//
// Currently unsupported types:
//
// ADSDATATYPEID.ADST_BIGTYPE;
// ADSDATATYPEID.ADST_REAL80;
// ADSDATATYPEID.ADST_VOID;
// ADSDATATYPEID.ADST_STRING
// ADSDATATYPEID.ADST_WSTRING

FUNCTION F_ParseToVariant : bool
VAR_INPUT
	adsTypeID  : ADSDATATYPEID;
	sValue		 : STRING;
END_VAR
VAR_IN_OUT
		var_data : ST_VARIANT;
END_VAR


	F_ParseToVariant:= TRUE;	
	
	CASE adsTypeID OF 
		
		ADSDATATYPEID.ADST_INT8:
			var_data.nI8 := STRING_TO_SINT(sValue);

		ADSDATATYPEID.ADST_UINT8:
			var_data.nUI8 := STRING_TO_USINT(sValue);
					
		ADSDATATYPEID.ADST_INT16:
			var_data.nI16 := STRING_TO_INT(sValue);
		
		ADSDATATYPEID.ADST_UINT16:
			var_data.nUI16 := STRING_TO_UINT(sValue);
						
		ADSDATATYPEID.ADST_INT32:
			var_data.nI32 := STRING_TO_DINT(sValue);

		ADSDATATYPEID.ADST_UINT32:
			var_data.nUI32 := STRING_TO_UDINT(sValue);
			
		ADSDATATYPEID.ADST_INT64:
			var_data.nI64 := STRING_TO_LINT(sValue);

		ADSDATATYPEID.ADST_UINT64:
			var_data.nUI64 := STRING_TO_ULINT(sValue);			

		ADSDATATYPEID.ADST_REAL32:
			var_data.fR32 := STRING_TO_REAL(sValue);
						
		ADSDATATYPEID.ADST_REAL64:
			var_data.fR64 := STRING_TO_LREAL(sValue);
			
		ADSDATATYPEID.ADST_BIT:
			var_data.nBit := INT_TO_BOOL(STRING_TO_INT(sValue));

		ELSE
			F_ParseToVariant:= FALSE;	
		END_CASE

END_FUNCTION

(* stored: Version 1.1.0.1, ProductVersion 3.1.4024.12
   POU F_ParseToVariant: Id {20cf5fb8-5dd5-47c0-90b2-4963bf0c31dd}, SpecialFunc None *)
